{attribute 'qualified_only'}
{attribute 'strict'}
TYPE E_TransportResponse :
(
	Accepted := 0,
	DivertLaneUnavailable := 1,
	LoadIdNotFound := 2,
	UnknownFailure := 11,
	NextLoadReady := 12,
	LateInduction := 13
);
END_TYPE

(* stored: Version 1.1.0.1, ProductVersion 3.1.4024.4
   EnumerationTextList E_TransportResponse: Id {f32ac88b-b9b5-4b8c-94a3-d148c71bd0e7} *)
